{attribute addProperty BoxType "EK1100-0000-0018"}
{attribute addProperty Id "Beckhoff_EP1xxxEK1122Beckhoff_EP1xxxEK1122_B7B205631214068719478253.5"}
{attribute addProperty CRC "3370633563"}
{attribute addProperty SizeInBites "12140"}
{attribute addProperty SizeInBytes "68719478253.5"}
TYPE Beckhoff_EP1xxx_C8E7C95B EXTENDS EK1100_179A0949 :
STRUCT
	{attribute addProperty Name "Beckhoff_EP1xxxEK1122"}
	Beckhoff_EP1xxxEK1122 : Beckhoff_EP1xxxEK1122_B7B20563;
END_STRUCT
END_TYPE

(* stored: Version 1.2.0.0, ProductVersion 3.1.4024.9
   DUT Beckhoff_EP1xxx_C8E7C95B: Id {575587e8-ca6e-414e-8699-356a6b336c1e} *)
